FUNCTION_BLOCK FB_MonetTelescopeControl EXTENDS FB_AltAzTelescopeControl IMPLEMENTS I_AltAzTelescope
VAR_INPUT
	fbFocus				: I_Focus;
	fbCovers			: I_MirrorCovers;
	fbBrake				: I_Brake;	
	fbHydraulics   		: I_Hydraulics;
	fbElevation			: REFERENCE TO FB_ElevationControl;
	fbAzimuth			: REFERENCE TO FB_AzimuthControl;
	fbDerotator			: REFERENCE TO FB_DerotatorControl;

	fbPointing			: REFERENCE TO FB_PointingModelForward;
	fbPointingInverse	: REFERENCE TO FB_PointingModelInversion;

	bBrakeClearing		: BOOL	:= TRUE;

	// M6: applied to every commanded elevation move (Goto/Home/Park/PowerOn/Slew, not
	// the computed tracking rate), NOT just _HomeTelescope despite the old name.
	// 5.0 deg/s confirmed correct on-site for MONETS; 10.0 was too fast.
	fElevationMoveVelocity : LREAL := 5.0;
END_VAR
VAR_OUTPUT
	fDerotatorSign		: LREAL := 1.0;	// derotator
	
	fElevationPointingOffset : LREAL;
	fAzimuthPointingOffset : LREAL;
	fElevationPointingOffset2 : LREAL;
	fAzimuthPointingOffset2 : LREAL;
	
	fRightAscensionCurrentSky: LREAL;
	fDeclinationCurrentSky: LREAL;

	fDerotatorVelocity	: LREAL;	// rotational velocity of the derotator
	fElevationVelocity	: LREAL;	// rotational velocity of the elevation
	fAzimuthVelocity	: LREAL;	// rotational velocity of the elevation
END_VAR
VAR
	// M1: internal (non-axis) errors from the Goto/Home/Slew state machines, latched
	// until bReset since bError/nErrorID are otherwise recomputed from the axes every
	// scan and would silently wipe these within the same cycle they're set in.
	bSoftwareError		: BOOL;
	nSoftwareErrorID	: UINT;
	SoftwareErrorEvent	: FB_EventLog;

	// #26 / ADR 0001 option 1: auto-clear a latched bInterrupted if nothing has been
	// requested for a while, since the normal arbitration path can never do it on its
	// own (bReady needs the axes enabled, axis enable needs bInterrupted already clear).
	// Visible, not silent: logged and counted, not just quietly cleared.
	bInterruptedIdle			: BOOL;
	tonInterruptedAutoClear		: TON;
	InterruptedAutoClearEvent	: FB_EventLog;
END_VAR
VAR PERSISTENT
	nInterruptedAutoClearCount	: UDINT;	// how many times auto-clear has fired, ever
END_VAR

// revert fDut1 (set via the Dut1 property, e.g. from an external time bridge over MQTT) to its
// safe 0.0 default if nothing fresh arrives for a while, instead of serving an arbitrarily
// stale UT1-UTC correction forever. FB_AltAzTelescopeControl's own body is never called (this FB
// doesn't call SUPER^() in its main body), so this has to live here rather than up there.
tonDut1Stale(IN := NOT bDut1Received, PT := T#10M);
bDut1Received := FALSE;
IF tonDut1Stale.Q THEN
	fDut1 := 0.0;
END_IF

// get the system time; fJd only follows the clock while the clock is valid (synced, see FB_AstroClock)
fbTime();
IF fbTime.bValid THEN
	fJd := DateTime2JD(fbTime.time_RTCEX2);
END_IF
fLst := CT2LST(telescopeConfig.longitude, fJd);

// without a trustworthy time nothing may be pointed or tracked: refuse through the normal stop path
IF NOT fbTime.bValid AND (bGoto OR bSlew OR bTrack) THEN
	bStop := TRUE;
END_IF

// set reset state either by hardware (key pressed) or by software (set by e.g. tcs)
rtrigReset(CLK := bReset);

IF bReset THEN
	bHorizonError := FALSE; // if reset, the bHorizonError can be switched off
	bSoftwareError := FALSE;
	
	// reset the stages of all statemachine methods
	bInterrupted := TRUE; 
	_HomeTelescope();
	_GotoTelescope();
	_SlewTelescope();
	_ParkTelescope();
	bInterrupted := FALSE;
END_IF

// get error ID, reset if bReset command is set
IF fbAzimuth.Error THEN
	nErrorID := fbAzimuth.nErrorID;
	IF bReset THEN
		fbAzimuth.Reset();
	END_IF
ELSIF fbElevation.bError THEN
	nErrorID := fbElevation.nErrorID;
	IF bReset THEN
		fbElevation.Reset();
	END_IF
ELSIF fbDerotator.bError THEN
	nErrorID := fbDerotator.nErrorID;
	IF bReset THEN
		fbDerotator.Reset();
	END_IF	
ELSIF fbFocus.Error THEN
	nErrorID := fbFocus.ErrorID;
	IF bReset THEN
		fbFocus.Reset();
	END_IF
ELSIF bSoftwareError THEN
	nErrorID := nSoftwareErrorID;
END_IF

// fSlewTime
fSlewTime :=  MAX(MAX(fbElevation.fSlewTime, fbAzimuth.fSlewTime), fbDerotator.fSlewTime);

bError := fbElevation.Error OR
		 fbAzimuth.bError OR
		 fbFocus.Error OR
		 fbDerotator.bError OR
		 bSoftwareError;
			
IF bError THEN
	bTrack := 	FALSE;
	bGoto := 	FALSE;
	bSlew := 	FALSE;
	fbElevation.Enable := FALSE;
	fbAzimuth.Enable := FALSE;
	fbDerotator.Enable := FALSE;
ELSE
	nErrorID := 0;
END_IF

IF fbElevation.bError THEN
	fbElevation.Enable := FALSE;
	fbAzimuth.Enable := FALSE;
	fbDerotator.Enable := FALSE;
	fbBrake.CloseBrake();
END_IF

eq2hor(
	ra := fRightAscension,
	dec := fDeclination,
	lon := telescopeConfig.longitude,
	lat := telescopeConfig.latitude,
	altitude := telescopeConfig.altitude,
	JD := fJd + fTimeOffset,
	dut1 := fDut1,
	refract_to_observed := TRUE,
	// refract := FALSE,
	alt => fElevationCalc,
	az => fAzimuthCalc,
	ha => fHourAngleCalc);

// apply pointing model
fbPointing(
	fAzimuth			:= fAzimuthCalc,
	fElevation			:= fElevationCalc,
	fAzimuthOffset		=> fAzimuthPointingOffset,
	fElevationOffset	=> fElevationPointingOffset
);
fElevationCalc := fElevationCalc + fElevationPointingOffset + fElevationOffset;
// F_AzimuthOffsetOnAxis: fAzimuthOffset / COS(elevation), bounded near the zenith (BROTLib#27)
fAzimuthCalc := fAzimuthCalc + fAzimuthPointingOffset + F_AzimuthOffsetOnAxis(fAzimuthOffset, fElevationCalc);

// calculate derotator position 
fDerotatorCalc := F_DerotatorPosition2(fAzimuthCalc, fElevationCalc, telescopeConfig.latitude, fDerotatorSign)  + fDerotatorOffset;

// calculate velocities
fDerotatorVelocity := F_Derotatorvelocity(fAzimuthCalc, fElevationCalc, telescopeConfig.latitude, fDerotatorSign);
fElevationVelocity := F_Elevationvelocity(fAzimuthCalc, telescopeConfig.latitude);
fAzimuthVelocity := F_Azimuthvelocity(fElevationCalc, fAzimuthCalc, telescopeConfig.latitude);

IF (fAzimuthCalc > 310.0 AND fAzimuthVelocity > 0.0) OR (fAzimuthCalc > 440.0) THEN
	fAzimuthCalc := fAzimuthCalc - 360.0;
ELSIF (fAzimuthCalc < 80.0 AND fAzimuthVelocity < 0.0) OR (fAzimuthCalc < -50.0) THEN
	fAzimuthCalc := fAzimuthCalc + 360.0;
END_IF

IF (fDerotatorCalc > 290.0 AND fDerotatorVelocity > 0.0) OR (fDerotatorCalc > 380.0) THEN
	fDerotatorCalc := fDerotatorCalc - 360.0;
ELSIF (fDerotatorCalc < 20.0 AND fDerotatorVelocity < 0.0) OR (fDerotatorCalc < -70.0) THEN
	fDerotatorCalc := fDerotatorCalc + 360.0;
END_IF

// get current coordinates	
fAzimuthCurrent := fbAzimuth.fActualPosition;
fElevationCurrent := fbElevation.fActualPosition;
fDerotatorCurrent := fbDerotator.fActualPosition;

// apply inverse pointing model
fbPointingInverse(
	fAzimuth			:= fAzimuthCurrent,
	fElevation			:= fElevationCurrent,
	fAzimuthOffset  	=> fAzimuthPointingOffset2,
	fElevationOffset	=> fElevationPointingOffset2
);
fAzimuthCurrentSky := fAzimuthCurrent - fAzimuthPointingOffset2;
fElevationCurrentSky := fElevationCurrent - fElevationPointingOffset2;

// add offsets
//fElevationCurrent := fElevationCurrentSky - fElevationOffset;
//fAzimuthCurrent := fAzimuthCurrentSky - fAzimuthOffset / COS(fElevationCalc * d2r);

// calculate equatorial coordinates
hor2eq(alt := fElevationCurrentSky - fElevationOffset,
		az := fAzimuthCurrentSky - F_AzimuthOffsetOnAxis(fAzimuthOffset, fElevationCurrent),	// M7: was fElevationCalc
		jd := fJd,
		dut1 := fDut1,
		lat := telescopeConfig.latitude,
		lon := telescopeConfig.longitude,
		altitude := telescopeConfig.altitude,
		alt_is_observed := TRUE,
		// refract := FALSE,
		ra => fRightAscensionCurrent,
		dec => fDeclinationCurrent,
		ha => fHourAngleCurrent);	// M13: was never assigned, HA_ICRS telemetry was stuck at 0.0
hor2eq(alt := fElevationCurrentSky,
		az := fAzimuthCurrentSky,
		jd := fJd,
		dut1 := fDut1,
		lat := telescopeConfig.latitude,
		lon := telescopeConfig.longitude,
		altitude := telescopeConfig.altitude,
		alt_is_observed := TRUE,
		ra => fRightAscensionCurrentSky,
		dec => fDeclinationCurrentSky);
	
// If the Telescope dips under the fHorizon (e.g. while tracking, stop and gohome)
IF fbElevation.Calibrated AND fElevationCurrent < (fHorizon+0.2) THEN
	IF NOT bStopped AND NOT bGoHome THEN
		bStop := TRUE;
	ELSE
		bGoHome := TRUE;
	END_IF
END_IF
		
tpPowerOnWarning(IN := bPower OR (NOT fbElevation.bEnable AND fbBrake.BrakeOpen), PT := T#250MS);

tonPowerTimeout(IN := TCS_command = E_TCSCommand.no_command AND NOT bIsParked, PT := T#12H);
tonCommandTimeout();
IF tonPowerTimeout.Q AND NOT bIsParked THEN
	bPark := TRUE;
END_IF
		
// #26 / ADR 0001 option 1: bInterrupted otherwise cannot clear itself once latched with
// nothing pending (see specs/design/telescopecontrol-command-arbitration.md); auto-clear
// after a few seconds of true idle (no error, nothing requested), logged and counted so
// it's visible rather than a silent recovery. TUNE PT if this fires too eagerly/late on
// site.
bInterruptedIdle := bInterrupted AND NOT bError AND
	NOT (bPower OR bPark OR bGoHome OR bGoto OR bSlew OR bTrack);
tonInterruptedAutoClear(IN := bInterruptedIdle, PT := T#5S);
IF tonInterruptedAutoClear.Q THEN
	bInterrupted := FALSE;
	nInterruptedAutoClearCount := nInterruptedAutoClearCount + 1;
END_IF
InterruptedAutoClearEvent(
	Trigger 		:= tonInterruptedAutoClear.Q,
	Level 			:= ADSLOG_MSGTYPE_WARN,
	FormatString 	:= 'bInterrupted auto-cleared after idle timeout (count: %s)',
	OnMessage 		:= UDINT_TO_STRING(nInterruptedAutoClearCount),
	Comm 			:= fbComm);

// set TCS_command according to state variables ordered by precedence
// Stop outranks everything, including a running power-on
IF bStop THEN
	bTrack := FALSE;
	
	// If the stop is during a power-on or a movement, reset the stage of the movement first
	IF bPower THEN
		bPower := FALSE;
		_PowerOn();
	END_IF
	IF bPark THEN
		bPark := FALSE;
		_ParkTelescope();
	ELSIF bGoto THEN
		bGoto := FALSE;
		_GotoTelescope();
	ELSIF bSlew THEN
		bSlew := FALSE;
		_SlewTelescope();
	ELSIF bGoHome THEN
		bGoHome := FALSE;
		_HomeTelescope();
	END_IF
	TCS_command := E_TCSCommand.stop;
	
ELSIF bPower THEN
	TCS_command := E_TCSCommand.poweron;
	
ELSIF bPark THEN
	bTrack := FALSE;
	// M2: emergency park bypasses the bReady/bBusy gating below entirely, since bReady
	// requires NOT bError and would otherwise make park unreachable during an error.
	IF bError THEN
		bInterrupted := FALSE;
		TCS_command := E_TCSCommand.park;
	// If lower presedence commands are ongoing, let them know they are interupted
	ELSIF bGoto OR bSlew OR bGoHome THEN
		bGoHome := FALSE;
		bGoto := FALSE;
		bSlew := FALSE;
		bInterrupted := TRUE;
		_HomeTelescope();
		_GotoTelescope();
		_SlewTelescope();

	ELSE
		IF bReady AND NOT bBusy THEN
			bInterrupted := FALSE;
			TCS_command := E_TCSCommand.park;
		END_IF
	END_IF
	
ELSIF bGoHome THEN
	bTrack := FALSE;
	// If lower presedence commands are ongoing, let them know they are interupted
	IF bGoto OR bSlew THEN
		bGoto := FALSE;
		bSlew := FALSE;
		bInterrupted := TRUE;
		_GotoTelescope();
		_SlewTelescope();
		
	ELSE
		IF bReady AND NOT bBusy AND bStopped THEN
			bInterrupted := FALSE;
			TCS_command := E_TCSCommand.gohome;
		END_IF
	END_IF
	
	
ELSIF bGoto THEN
	bTrack := FALSE;
	// If lower presedence commands are ongoing, let them know they are interupted
	IF bSlew THEN
		bSlew := FALSE;
		bInterrupted := TRUE;
		_SlewTelescope();
	ELSE
		IF bReady AND NOT bBusy THEN
			bInterrupted := FALSE;
			TCS_command := E_TCSCommand.goto;
		END_IF
	END_IF
		
ELSIF bSlew THEN
	bTrack := FALSE;
	IF bReady AND NOT bBusy THEN
		TCS_command := E_TCSCommand.slew;
	END_IF
	
ELSIF bTrack THEN
	IF bReady AND NOT bBusy THEN
		TCS_command := E_TCSCommand.track;
	END_IF
	
ELSE
	TCS_command := E_TCSCommand.no_command;
	fbElevation.bMoveAxis := FALSE;
	fbAzimuth.bMoveAxis := FALSE;
	fbDerotator.bMoveAxis := FALSE;
	fbElevation.bTracking := FALSE;
	fbAzimuth.bTracking := FALSE;
	fbDerotator.bTracking := FALSE;
END_IF

IF TCS_command = E_TCSCommand.poweron THEN
	_PowerOn();
	tonCommandTimeout(IN := TCS_command = E_TCSCommand.poweron, PT := T#12H);
	TCSCTOEvent.OnMessage := 'POWER';
ELSIF TCS_command = E_TCSCommand.stop THEN
	_StopTelescope();
	tonCommandTimeout(IN := TCS_command = E_TCSCommand.stop, PT := T#2S);
	TCSCTOEvent.OnMessage := 'STOP';
ELSIF TCS_command = E_TCSCommand.park THEN
	_ParkTelescope();
	tonCommandTimeout(IN := TCS_command = E_TCSCommand.park, PT := T#2M);
	TCSCTOEvent.OnMessage := 'PARK';
ELSIF TCS_command = E_TCSCommand.gohome THEN
	_HomeTelescope();
	tonCommandTimeout(IN := TCS_command = E_TCSCommand.gohome, PT := T#2M);
	TCSCTOEvent.OnMessage := 'GOHOME';
ELSIF TCS_command = E_TCSCommand.goto THEN
	_GotoTelescope();
	tonCommandTimeout(IN := TCS_command = E_TCSCommand.goto, PT := T#2M);
	TCSCTOEvent.OnMessage := 'GOTO';
ELSIF TCS_command = E_TCSCommand.slew THEN
	_SlewTelescope();
	tonCommandTimeout(IN := TCS_command = E_TCSCommand.slew, PT := T#2M);
	TCSCTOEvent.OnMessage := 'SLEW';
ELSIF TCS_command = E_TCSCommand.track THEN
	_TrackTelescope();
	tonCommandTimeout(IN := TCS_command = E_TCSCommand.track, PT := T#12H);
	TCSCTOEvent.OnMessage := 'TRACK';
ELSE
	// disable command timeout
	tonCommandTimeout(IN := FALSE);
	TCSCTOEvent.OnMessage := 'NOCOMMAND';
END_IF
 
bSlewing := NOT bTracking AND (fbElevation.fbAxis.InMotion OR fbElevation.fbAxis.InRamp OR
			fbAzimuth.fbAxis.InMotion OR fbAzimuth.fbAxis.InRamp OR
			fbDerotator.fbAxis.InMotion OR fbDerotator.fbAxis.InRamp);

// signal must be stable for 5500MS
tonTrackingDelay(in := fbElevation.fbAxis.isTracking AND 
			fbAzimuth.fbAxis.isTracking AND
			fbDerotator.fbAxis.isTracking,PT :=T#5500MS, Q => bTracking);
			
bStopped :=  (NOT fbElevation.bEnable OR fbElevation.fbAxis.StandStill) AND 
			(NOT fbAzimuth.bEnable OR fbAzimuth.fbAxis.StandStill) AND
			(NOT fbDerotator.bEnable OR fbDerotator.fbAxis.StandStill);
			
bHomed := fbElevation.Calibrated AND
			fbAzimuth.Calibrated AND
			fbFocus.Calibrated AND
			fbDerotator.Calibrated;
			
bReady := bHomed AND 
	fbCovers.Opened AND 
	fbElevation.bEnable AND
	fbAzimuth.bEnable AND
	fbDerotator.bEnable AND fbBrake.BrakeOpen AND 
    NOT bError;

bBusy := fbElevation.fbAxis.Busy OR
		fbAzimuth.fbAxis.Busy OR
		fbDerotator.fbAxis.Busy OR
		fbFocus.Busy;

(* STATUS STATES*)
//fReadyState (see also _PowerOn and _ParkTelescope calls above)
IF bError THEN
	fReadyState := -1.0;
ELSIF bPower THEN
	fReadyState := 0.7;
ELSIF bIsParked THEN
	fReadyState := 0.0;
ELSIF bPark THEN
	fReadyState := 0.3;
ELSIF bReady THEN
	fReadyState := 1.0;	
ELSE
	fReadyState := -2.0;	
END_IF

//MotionState
IF bStopped THEN
	nMotionState := 0;
ELSIF bSlewing OR bBusy THEN
	nMotionState := 1;
ELSIF bTracking THEN
	nMotionState := 8;
END_IF

// unset the STOP command if telescope is already stopped
IF bStopped THEN
	bStop := FALSE;
END_IF
	
IF NOT bError THEN
	bReset := FALSE;
END_IF

IF bEstopTriggered THEN
	fbElevation.Enable := FALSE;
	fbAzimuth.Enable := FALSE;
	fbDerotator.Enable := FALSE;
END_IF

// send telemetry
IF bSlewing OR bTrack OR bTracking THEN
	tonMQTTTimer.PT := T#500MS; // M13: was "every second", actually twice a second while moving
ELSE
	tonMQTTTimer.PT := T#1000MS; // M13: was "every five seconds", actually every second otherwise
END_IF
tonMQTTTimer(IN:=TRUE);
IF tonMQTTTimer.Q THEN
	tonMQTTTimer(IN:=FALSE);
	_SendTelemetry();
END_IF


(* Event function blocks start here. *)
TCSpowerEvent(	Trigger := bPowerFailure, 
				Level := ADSLOG_MSGTYPE_ERROR,
				FormatString := 'power %s',
				//OnMessage := 'Failure',
				OffMessage := 'OK', 
				Comm := fbComm);

TCSgohomeEvent(	Trigger := bGoHome, 
				Level := ADSLOG_MSGTYPE_HINT,
				FormatString := 'GOHOME %s',
				OnMessage := 'commencing',
				OffMEssage := 'completed', 
				Comm := fbComm);
TCSparkEvent(	Trigger := bPark, 
				Level := ADSLOG_MSGTYPE_HINT,
				FormatString := 'PARK %s',
				OnMessage := 'commencing',
				OffMEssage := 'completed', 
				Comm := fbComm);
TCSgotoEvent(	Trigger := bGoto, 
				Level := ADSLOG_MSGTYPE_HINT,
				FormatString := 'GOTO %s',
				OnMessage := 'commencing',
				OffMEssage := 'completed', 
				Comm := fbComm);
TCStrackEvent(	Trigger := bTrack, 
				Level := ADSLOG_MSGTYPE_HINT,
				FormatString := 'TRACK %s',
				OnMessage := 'commencing',
				OffMEssage := 'completed', 
				Comm := fbComm);
TCSstopEvent(	Trigger := bStop, 
				Level := ADSLOG_MSGTYPE_WARN,
				FormatString := 'STOP %s',
				OnMessage := 'commencing',
				OffMEssage := 'completed',
				OffLevel := ADSLOG_MSGTYPE_HINT, 
				Comm := fbComm);
TCStargetHorizonEvent(	Trigger := fElevationCalc<fHorizon,
				Level := ADSLOG_MSGTYPE_WARN,
				FormatString := '%s',
				OnMessage := 'Target below safe horizon',
				OffMEssage := '', 
				Comm := fbComm);
TCSreadyEvent(	Trigger := bPower AND bReady, 
				Level := ADSLOG_MSGTYPE_HINT,
				FormatString := '%s',
				OnMessage := 'STELLA1 startup finished', 
				Comm := fbComm);
TCSCTOEvent(	Trigger := tonCommandTimeout.Q,
				Level := ADSLOG_MSGTYPE_WARN,
				FormatString := 'A timeout occurred during %s command!',
				OnMessage := 'NOCOMMAND',
				Comm := fbComm);
SoftwareErrorEvent(	Trigger := bSoftwareError,
				Level := ADSLOG_MSGTYPE_ERROR,
				FormatString := 'Internal command error, ID: %s',
				OnMessage := UINT_TO_STRING(nSoftwareErrorID),
				OffMessage := 'cleared',
				OffLevel := ADSLOG_MSGTYPE_HINT,
				Comm := fbComm);

METHOD PRIVATE _GotoTelescope : USINT
VAR_INPUT
END_VAR
VAR
	GoToEvent		: FB_Eventlog;
	commandTimeout	: TON;
END_VAR
VAR_STAT
	nStage			: USINT := 0;
	nLastStage		: USINT := 101;
END_VAR
_GotoTelescope := nStage;
commandTimeout(IN := nStage < 100, PT := T#600S);
IF commandTimeout.Q THEN
	bError := TRUE;
	nErrorID := 16#10;
	bSoftwareError := TRUE;
	nSoftwareErrorID := 16#10;
	bGoto := FALSE;
	nStage := 0;
	RETURN;
END_IF

IF fElevationCalc<2.0 THEN
	bError := TRUE;
	nErrorID := 16#15;
	bSoftwareError := TRUE;
	nSoftwareErrorID := 16#15;
	bGoto := FALSE;
	nStage := 0;
	RETURN;
END_IF

// M7: near zenith COS(elevation) -> 0, so any nonzero fAzimuthOffset blows up into a
// huge azimuth (see the offset divisions elsewhere in this FB). 89.5 matches the
// existing tracking cutoff (_TrackTelescope: fElevationCurrent > 89.5).
IF fElevationCalc>89.5 THEN
	bError := TRUE;
	nErrorID := 16#16;
	bSoftwareError := TRUE;
	nSoftwareErrorID := 16#16;
	bGoto := FALSE;
	nStage := 0;
	RETURN;
END_IF

IF bReset OR bError OR bInterrupted THEN
	nStage := 0;
	RETURN;
END_IF

CASE nStage OF
	0:	
		IF bReady AND NOT bBusy THEN
			nStage := 10;
		END_IF
	10:
		IF fbElevation.Tracking = TRUE OR fbAzimuth.Tracking = TRUE OR fbDerotator.Tracking = TRUE THEN
			fbElevation.Tracking := FALSE;
			fbAzimuth.Tracking := FALSE;
			fbDerotator.Tracking := FALSE;
		ELSE
			nStage := 25;
		END_IF				
	25:	
		fbElevation.Position := fElevationCalc;
		fbAzimuth.Position := fAzimuthCalc;
		fbDerotator.Position := fDerotatorCalc;
		fbDerotator.Velocity := 10.0;
		fbElevation.Velocity := fElevationMoveVelocity;
		fbAzimuth.Velocity := 10.0;
		
		fbElevation.MoveAxis := TRUE;
		fbAzimuth.MoveAxis := TRUE;
		fbDerotator.MoveAxis := TRUE;
		IF fbElevation.Busy AND
			fbAzimuth.Busy AND
			fbDerotator.Busy THEN
				nStage := 50;
		END_IF
	50:
		IF NOT fbElevation.Busy AND fbElevation.MoveDone THEN
			fbElevation.MoveAxis := FALSE;
		END_IF
		IF NOT fbAzimuth.Busy AND fbAzimuth.MoveDone THEN
			fbAzimuth.MoveAxis := FALSE;
		END_IF
		IF NOT fbDerotator.Busy AND fbDerotator.MoveDone THEN
			fbDerotator.MoveAxis := FALSE;
		END_IF
		IF NOT fbElevation.MoveAxis AND 
           NOT fbAzimuth.MoveAxis AND 
		   NOT fbDerotator.MoveAxis THEN
		   nStage := 75;
		END_IF
	75:
		IF NOT bSlewing AND bStopped THEN // all axis standstill
			nStage := 100;
		END_IF
	100:
		fbElevation.MoveAxis := FALSE;
		fbAzimuth.MoveAxis := FALSE;
		fbDerotator.MoveAxis := FALSE;
		fAzimuth := fAzimuthCalc;
		fElevation := fElevationCalc;
		bGoto := FALSE;
		// enable automatic tracking
		bTrack := bAutoTrack;
		nStage := 0;
END_CASE
GoToEvent(Trigger := nStage > nLastStage, FormatString := 'GoTo progress: %s', OnMessage := USINT_TO_STRING(nStage), comm := fbComm);
nLastStage := nStage;
END_METHOD

METHOD PRIVATE _HomeTelescope : BOOL
VAR_INPUT
END_VAR
VAR
    HomeEvent        : FB_Eventlog;
    commandTimeout    : TON;
END_VAR
// reset/interrupt aborts the homing without moving anything, like the other stage methods
IF bReset OR bError OR bInterrupted THEN
    commandTimeout(IN := FALSE);
    RETURN;
END_IF

commandTimeout(IN := NOT _HomeTelescope, PT := T#600S);
IF commandTimeout.Q THEN
    bError := TRUE;
    nErrorID := 16#30;
    bSoftwareError := TRUE;
    nSoftwareErrorID := 16#30;
    _HomeTelescope :=TRUE;
END_IF

// only move while a home command is active (Stop/Park/Reset call this with bGoHome cleared to abort it)
IF bGoHome AND bReady AND bStopped AND NOT bBusy AND NOT bTracking THEN
    fbElevation.Velocity := fElevationMoveVelocity;
    fbElevation.Position := telescopeConfig.elevationHome;
    fbElevation.MoveAxis := TRUE;
    fbAzimuth.Velocity := 10.0;
    fbAzimuth.Position := telescopeConfig.azimuthHome;
    fbAzimuth.MoveAxis := TRUE;
    fbDerotator.Velocity := 10.0;
    fbDerotator.Position := telescopeConfig.derotatorHome;
    fbDerotator.MoveAxis := TRUE;    
END_IF

IF fbElevation.MoveDone AND 
    fbAzimuth.MoveDone AND 
    fbDerotator.MoveDone THEN
    bGoHome := FALSE;
    fElevation := fElevationCurrent;
    fAzimuth := fAzimuthCurrent;
    _HomeTelescope := TRUE;
ELSE
    _HomeTelescope := FALSE;
END_IF

HomeEvent(Trigger := _HomeTelescope, 
            Level := ADSLOG_MSGTYPE_HINT,
            FormatString := '%s',
            OnMessage := 'Telescope is homed.', comm := fbComm);
END_METHOD

METHOD PRIVATE _ParkTelescope : USINT
VAR_INPUT
END_VAR
VAR
	ParkEvent	: FB_Eventlog;
	rtrigError	: R_TRIG;	// M2: reset the stage only on the rising edge of bError, not every scan
END_VAR
VAR_STAT
	nStage		: USINT := 0;
	nLastStage	: USINT := 101;
END_VAR
_ParkTelescope := nStage;
IF bReset OR bStop OR bInterrupted THEN
	nStage := 0;
	RETURN;
END_IF
// M2: bError does NOT return early here, unlike the other state machines: stage 0's
// "emergency park" branch below is the safe-state response to bError and must run.
// Only force the stage back to 0 on the rising edge, so the emergency branch can still
// progress through its own stages (80 -> 100) on later scans while bError stays TRUE.
rtrigError(CLK := bError);
IF rtrigError.Q THEN
	nStage := 0;
END_IF
IF bIsParked THEN
	nStage := 100;
END_IF
CASE nStage OF
	0: 
		bGoHome := 	FALSE;
		bTrack := 	FALSE;
		bGoto := 	FALSE;
		bSlew := 	FALSE;
		fbFocus.Position := telescopeConfig.focusPark;
		IF bError THEN // emergency park
			fbBrake.CloseBrake();
			fbElevation.Enable := FALSE;
			fbAzimuth.Enable := FALSE;
			fbDerotator.Enable := FALSE;	
			fbCovers.Close();	
			nStage := 80;
		ELSE
			nStage := 10;
		END_IF
	10:
		IF fbElevation.Tracking = TRUE OR fbAzimuth.Tracking = TRUE OR fbDerotator.Tracking = TRUE THEN
			fbElevation.Tracking := FALSE;
			fbAzimuth.Tracking := FALSE;
			fbDerotator.Tracking := FALSE;
		ELSE
			nStage := 20;
		END_IF		
	20:
		fbElevation.Position := telescopeConfig.elevationPark;
		fbElevation.Velocity := fElevationMoveVelocity;
		fbElevation.MoveAxis := TRUE;
		fbAzimuth.Position := telescopeConfig.azimuthPark;
		fbAzimuth.Velocity := 10;
		fbAzimuth.MoveAxis := TRUE;
		fbDerotator.Position := telescopeConfig.derotatorPark;
		fbDerotator.Velocity := 10.0;
		fbDerotator.MoveAxis := TRUE;
		IF fbElevation.Busy AND
			fbAzimuth.Busy AND
			fbDerotator.Busy THEN
				nStage := 40;
		END_IF
	40:
		IF fbElevation.MoveDone THEN
			fbElevation.MoveAxis := FALSE;
		END_IF
		IF fbAzimuth.MoveDone THEN
			fbAzimuth.MoveAxis := FALSE;
		END_IF
		IF fbDerotator.MoveDone THEN
			fbDerotator.MoveAxis := FALSE;
		END_IF
		IF NOT bSlewing THEN // all axis standstill
			nStage := 60;
		END_IF
	60:
		IF NOT fbElevation.Enable AND NOT fbAzimuth.Enable AND NOT fbDerotator.Enable THEN
			nStage := 80;
		END_IF

		IF bStopped THEN
			fbElevation.Enable := FALSE;
			fbAzimuth.Enable := FALSE;
			fbDerotator.Enable := FALSE;
		END_IF
		
		fbElevation.bMoveAxis := FALSE;
		fbAzimuth.bMoveAxis := FALSE;
		fbDerotator.bMoveAxis := FALSE;
	80:
		IF fbElevation.Enable OR fbAzimuth.Enable OR fbDerotator.Enable THEN
			nStage := 60;
		END_IF
		IF NOT fbBrake.BrakeOpen THEN
			fbCovers.Close();
			fbHydraulics.Enable := FALSE;
		END_IF
		IF fbCovers.Closed THEN
			nStage := 100;
		END_IF
	100:
			bIsParked := TRUE;
			bPark := FALSE;
			_ParkTelescope := 100;
			nStage := 0;	
END_CASE
ParkEvent(Trigger := nStage > nLastStage, FormatString := 'Parking progress: %s', OnMessage := USINT_TO_STRING(nStage), comm := fbComm);
nLastStage := nStage;
END_METHOD

METHOD PRIVATE _PowerOn : BOOL
VAR_INPUT
END_VAR
VAR_STAT
	nStage		: USINT := 0;
	nLastStage	: USINT := 101;
END_VAR
IF NOT bBrakeClearing THEN
	bPowerFailure := TRUE;
	TCSpowerEvent.OnMessage := 'failure: brake clearing not set';
	bPower := FALSE;
ELSIF bError THEN
	bPowerFailure := TRUE;
	TCSpowerEvent.OnMessage := 'Generic error during power on occurred.';
	bPower := FALSE;
ELSE
	bPowerFailure := FALSE;		
END_IF

IF bReset OR bError OR bStop OR bInterrupted THEN
	nStage := 0;
	// abort without leaving the last written axis commands set
	fbElevation.MoveAxis := FALSE;
	fbElevation.HomeAxis := FALSE;
	fbAzimuth.MoveAxis := FALSE;
	fbAzimuth.HomeAxis := FALSE;
	fbDerotator.MoveAxis := FALSE;
	fbDerotator.HomeAxis := FALSE;
	fbFocus.HomeAxis := FALSE;
	RETURN;
END_IF

CASE nStage OF
	0:
		_PowerOn := FALSE;
		// COVER MUST BE OPENED FOR A SUCCESSFUL WAKE & SHAKE COMMAND!
		// unconditional by design: does not consult bCoverAutoOpen (see CoverAutoOpen.Set)
		fbCovers.Open();
		IF bMainReady AND fbCovers.Opened THEN
			nStage := 10;
		END_IF
		
	10:
		fbElevation.Enable := TRUE;
		fbAzimuth.Enable := TRUE;
		fbDerotator.Enable := TRUE;
		
		IF fbElevation.Ready AND NOT fbElevation.Calibrated THEN
			fbElevation.HomeAxis := TRUE;
		END_IF
		
		IF fbAzimuth.Ready AND NOT fbAzimuth.Calibrated THEN
			fbAzimuth.HomeAxis := TRUE;
		END_IF
		
		// enable derotator
		IF fbElevation.Ready THEN
			fbDerotator.HomeAxis := fbDerotator.Ready AND NOT fbDerotator.Calibrated;
		END_IF
		
		// start calibration of focus after elevation has been calibrated
		// this avoids imbalance by the M2 mirror on the elvation during its calibration
		IF fbElevation.Calibrated AND NOT fbFocus.Calibrated THEN
			fbFocus.Enable := TRUE;
			fbFocus.HomeAxis := TRUE;
		END_IF
	
		IF fbCovers.Opened AND fbElevation.Calibrated AND fbAzimuth.Calibrated AND fbDerotator.Calibrated AND fbFocus.Calibrated AND
			bReady AND bStopped AND NOT bBusy AND NOT bTracking THEN
			nStage := 30;
		END_IF
		
	30:
		fbElevation.Velocity := fElevationMoveVelocity;
		fbElevation.Position := telescopeConfig.elevationHome;
		fbElevation.MoveAxis := TRUE;
		fbAzimuth.Velocity := 10.0;
		fbAzimuth.Position := telescopeConfig.azimuthHome;
		fbAzimuth.MoveAxis := TRUE;
		fbDerotator.Velocity := 10.0;
		fbDerotator.Position := telescopeConfig.derotatorHome;
		fbDerotator.MoveAxis := TRUE;	
		
		IF fbElevation.MoveDone AND 
			fbAzimuth.MoveDone AND 
			fbDerotator.MoveDone THEN
			nStage := 100;
		END_IF
			
	100:
		bPower := FALSE;
		fElevation := fElevationCurrent;
		fAzimuth := fAzimuthCurrent;
		_PowerOn := TRUE;
		bIsParked := FALSE;
		nStage := 0;
	
END_CASE
END_METHOD

METHOD _SendTelemetry : BOOL
VAR_INPUT
END_VAR
SUPER^._PublishTelemetry();

fbComm.Publish('telescope', 'dome', 'TELESCOPE.READY_STATE',	LREAL_TO_STRING(fReadyState));
fbComm.Publish('telescope', 'dome', 'TELESCOPE.MOTION_STATE',	LREAL_TO_STRING(nMotionState));
fbComm.Publish('telescope', 'dome', 'TELESCOPE.INTERRUPTED_AUTO_CLEAR_COUNT', UDINT_TO_STRING(nInterruptedAutoClearCount));

// INFO, CONFIG.MOUNTOPTIONS/MOUNT, STATUS.GLOBAL, OBJECT.INSTRUMENTAL.ALT/AZ and the static
// OBJECT.EQUATORIAL.EPOCH/EQUINOX/RA_PM/DEC_PM/RA_RATE/DEC_RATE fields used to be republished
// here too, byte-identical to what SUPER^._PublishTelemetry() above already sends under the same
// field names from the same source variables -- removed as pure duplication (#22).
//
// OBJECT.EQUATORIAL.RA_ICRS/DEC_ICRS kept even though pybrotlib's schema (the Python MQTT
// consumer, BROTLib/pyBROT src/pybrotlib/telemetry.py) has no such field under
// object.equatorial -- only object.equatorial.ra/dec, which SUPER already publishes with the
// same value -- so this specific publish looks like dead weight for that consumer. Not removing
// it here anyway: Telegraf/InfluxDB ingests the raw MQTT line independent of pybrotlib's schema,
// so something else could still depend on this exact field name landing in Influx. (For contrast,
// POSITION.EQUATORIAL.RA_ICRS/DEC_ICRS -- a different field, published further down -- *is* in
// pybrotlib's schema and is a real, actively consumed field.)
//
// OBJECT.HORIZONTAL.ALT/AZ below is also kept even though SUPER publishes those same field names:
// SUPER's version is conditional on bSlew (fElevation/fAzimuth vs fElevationCalc/fAzimuthCalc);
// this unconditional republish runs after it and is what has actually been on the wire -- changing
// that is a behavior change, not a dedup.

// EQUATORIAL
// all angles in the telemetry are degrees, RA included, like the rightascension command (BROTLib#37)
fbComm.Publish('telescope', 'dome', 'OBJECT.EQUATORIAL.RA_ICRS', LREAL_TO_STRING(fRightAscension));
fbComm.Publish('telescope', 'dome', 'OBJECT.EQUATORIAL.DEC_ICRS', LREAL_TO_STRING(fDeclination));

// HORIZONTAL
fbComm.Publish('telescope', 'dome', 'OBJECT.HORIZONTAL.ALT', LREAL_TO_STRING(fElevationCalc));
fbComm.Publish('telescope', 'dome', 'OBJECT.HORIZONTAL.AZ', LREAL_TO_STRING(fAzimuthCalc));

(* POINTING *)
fbComm.Publish('telescope', 'dome', 'POINTING.SLEWTIME', LREAL_TO_STRING(fSlewtime));
fbComm.Publish('telescope', 'dome', 'POINTING.OFFSETS.ALT', LREAL_TO_STRING(fElevationPointingOffset));
fbComm.Publish('telescope', 'dome', 'POINTING.OFFSETS.AZ', LREAL_TO_STRING(fAzimuthPointingOffset));

(*POSITION*)
//LOCAL
fbComm.Publish('telescope', 'dome', 'POSITION.LOCAL.SIDEREAL_TIME', LREAL_TO_STRING(fLst));
fbComm.Publish('telescope', 'dome', 'POSITION.LOCAL.JD', LREAL_TO_STRING(fJd));
fbComm.Publish('telescope', 'dome', 'POSITION.LOCAL.LATITUDE', LREAL_TO_STRING(telescopeConfig.latitude));
fbComm.Publish('telescope', 'dome', 'POSITION.LOCAL.LONGITUDE', LREAL_TO_STRING(telescopeConfig.longitude));
fbComm.Publish('telescope', 'dome', 'POSITION.LOCAL.HEIGHT', LREAL_TO_STRING(telescopeConfig.altitude));

// INSTRUMENTAL
// > ALT
// POWER_STATE
IF fbElevation.Enable THEN
	fbComm.Publish('telescope', 'dome', 'POSITION.INSTRUMENTAL.ALT.POWER_STATE', '1.0');
ELSE
	fbComm.Publish('telescope', 'dome', 'POSITION.INSTRUMENTAL.ALT.POWER_STATE', '0.0');
END_IF
//REFERENCED
IF fbElevation.Calibrated THEN
	fbComm.Publish('telescope', 'dome', 'POSITION.INSTRUMENTAL.ALT.REFERENCED', '1.0');
ELSE
	fbComm.Publish('telescope', 'dome', 'POSITION.INSTRUMENTAL.ALT.REFERENCED', '0.0');
END_IF
//ERROR_STATE
IF fbElevation.Error THEN
	fbComm.Publish('telescope', 'dome', 'POSITION.INSTRUMENTAL.ALT.ERROR_STATE', UDINT_TO_STRING(fbElevation.ErrorID));
ELSE
	fbComm.Publish('telescope', 'dome', 'POSITION.INSTRUMENTAL.ALT.ERROR_STATE', '0');
END_IF
//MOTION_STATE
IF fbElevation.Busy THEN
	IF fbElevation.isTracking THEN
		fbComm.Publish('telescope', 'dome', 'POSITION.INSTRUMENTAL.ALT.MOTION_STATE', '8');
	ELSE
		fbComm.Publish('telescope', 'dome', 'POSITION.INSTRUMENTAL.ALT.MOTION_STATE', '1');
	END_IF
ELSE
	fbComm.Publish('telescope', 'dome', 'POSITION.INSTRUMENTAL.ALT.MOTION_STATE', '0');
END_IF
fbComm.Publish('telescope', 'dome', 'POSITION.INSTRUMENTAL.ALT.REALPOS', LREAL_TO_STRING(fElevationCurrent-fElevationOffset));
fbComm.Publish('telescope', 'dome', 'POSITION.INSTRUMENTAL.ALT.CURRPOS', LREAL_TO_STRING(fElevationCurrent));
fbComm.Publish('telescope', 'dome', 'POSITION.INSTRUMENTAL.ALT.TARGETPOS', LREAL_TO_STRING(fbElevation.Position));
fbComm.Publish('telescope', 'dome', 'POSITION.INSTRUMENTAL.ALT.CURRSPEED', LREAL_TO_STRING(fbElevation.Velocity));
fbComm.Publish('telescope', 'dome', 'POSITION.INSTRUMENTAL.ALT.TARGETDISTANCE', LREAL_TO_STRING(ABS(fElevationCurrent-fbElevation.Position)));
fbComm.Publish('telescope', 'dome', 'POSITION.INSTRUMENTAL.ALT.OFFSET', LREAL_TO_STRING(fElevationOffset));

// > AZ
// POWER_STATE
IF fbAzimuth.Enable THEN
	fbComm.Publish('telescope', 'dome', 'POSITION.INSTRUMENTAL.AZ.POWER_STATE', '1.0');
ELSE
	fbComm.Publish('telescope', 'dome', 'POSITION.INSTRUMENTAL.AZ.POWER_STATE', '0.0');
END_IF
//REFERENCED
IF fbAzimuth.Calibrated THEN
	fbComm.Publish('telescope', 'dome', 'POSITION.INSTRUMENTAL.AZ.REFERENCED', '1.0');
ELSE
	fbComm.Publish('telescope', 'dome', 'POSITION.INSTRUMENTAL.AZ.REFERENCED', '0.0');
END_IF
//ERROR_STATE
IF fbAzimuth.Error THEN
	fbComm.Publish('telescope', 'dome', 'POSITION.INSTRUMENTAL.AZ.ERROR_STATE', UDINT_TO_STRING(fbAzimuth.ErrorID));
ELSE
	fbComm.Publish('telescope', 'dome', 'POSITION.INSTRUMENTAL.AZ.ERROR_STATE', '0');
END_IF
//MOTION_STATE
IF fbAzimuth.Busy THEN
	IF fbAzimuth.isTracking THEN
		fbComm.Publish('telescope', 'dome', 'POSITION.INSTRUMENTAL.AZ.MOTION_STATE', '8');
	ELSE
		fbComm.Publish('telescope', 'dome', 'POSITION.INSTRUMENTAL.AZ.MOTION_STATE', '1');
	END_IF
ELSE
	fbComm.Publish('telescope', 'dome', 'POSITION.INSTRUMENTAL.AZ.MOTION_STATE', '0');
END_IF

fbComm.Publish('telescope', 'dome', 'POSITION.INSTRUMENTAL.AZ.CURRPOS', LREAL_TO_STRING(fAzimuthCurrent));
fbComm.Publish('telescope', 'dome', 'POSITION.INSTRUMENTAL.AZ.REALPOS', LREAL_TO_STRING(fAzimuthCurrent-F_AzimuthOffsetOnAxis(fAzimuthOffset, fElevationCurrent)));	// M7: was fElevation (stale)
fbComm.Publish('telescope', 'dome', 'POSITION.INSTRUMENTAL.AZ.TARGETPOS', LREAL_TO_STRING(fbAzimuth.Position));
fbComm.Publish('telescope', 'dome', 'POSITION.INSTRUMENTAL.AZ.CURRSPEED', LREAL_TO_STRING(fbAzimuth.Velocity));
fbComm.Publish('telescope', 'dome', 'POSITION.INSTRUMENTAL.AZ.TARGETDISTANCE', LREAL_TO_STRING(ABS(fAzimuthCurrent-fbAzimuth.Position)));
fbComm.Publish('telescope', 'dome', 'POSITION.INSTRUMENTAL.AZ.OFFSET', LREAL_TO_STRING(fAzimuthOffset));


(*HORIZONTAL*)
fbComm.Publish('telescope', 'dome', 'POSITION.HORIZONTAL.ALT', LREAL_TO_STRING(fElevationCurrentSky));
fbComm.Publish('telescope', 'dome', 'POSITION.HORIZONTAL.AZ', LREAL_TO_STRING(fAzimuthCurrentSky));
//fbComm.Publish('telescope', 'dome', 'POSITION.HORIZONTAL.DOME', LREAL_TO_STRING(fbDome.Position));

(*EQUITORIAL*)
fbComm.Publish('telescope', 'dome', 'POSITION.EQUATORIAL.RA_ICRS', LREAL_TO_STRING(fRightAscensionCurrent));	// degrees (BROTLib#37)
fbComm.Publish('telescope', 'dome', 'POSITION.EQUATORIAL.HA_ICRS', LREAL_TO_STRING(fHourAngleCurrent));
fbComm.Publish('telescope', 'dome', 'POSITION.EQUATORIAL.DEC_ICRS', LREAL_TO_STRING(fDeclinationCurrent));
END_METHOD

METHOD PRIVATE _SlewTelescope : USINT
VAR_INPUT
END_VAR
VAR
	SlewEvent:	FB_Eventlog;
	command_timeout: TON;
END_VAR
VAR_STAT
	nStage:		USINT := 0;
	nLastStage:	USINT := 101;
END_VAR
_SlewTelescope := nStage;
command_timeout(IN := nStage < 100, PT := T#600S);
IF command_timeout.Q THEN
	bError := TRUE;
	nErrorID := 16#40;
	bSoftwareError := TRUE;
	nSoftwareErrorID := 16#40;
	bSlew := FALSE;
	nStage := 0;
	RETURN;
END_IF
IF bReset OR bError OR bInterrupted THEN
	nStage := 0;
	RETURN;
END_IF
CASE nStage OF
	0:	
		IF bReady AND bStopped AND NOT bBusy AND NOT bTracking THEN
			nStage := 10;
		END_IF
	10:
		IF fbElevation.Tracking = TRUE OR fbAzimuth.Tracking = TRUE OR fbDerotator.Tracking = TRUE THEN
			fbElevation.Tracking := FALSE;
			fbAzimuth.Tracking := FALSE;
			fbDerotator.Tracking := FALSE;
		ELSE
			nStage := 25;
		END_IF				
	25:
		fbPointing(
			fAzimuth			:= fAzimuth,
			fElevation			:= fElevation,
			fAzimuthOffset		=> fAzimuthPointingOffset,
			fElevationOffset	=> fElevationPointingOffset
		);	
		fbElevation.Position := fElevation + fElevationPointingOffset + fElevationOffset;
		fbElevation.Velocity := fElevationMoveVelocity;
		fbElevation.MoveAxis := TRUE;
		fbAzimuth.Position := fAzimuth + fAzimuthPointingOffset + F_AzimuthOffsetOnAxis(fAzimuthOffset, fElevation);	// M7: was fElevationCalc, mismatched with fAzimuth above
		fbAzimuth.Velocity := 10.0;
		fbAzimuth.MoveAxis := TRUE;
		fbDerotator.Position := fElevation + fDerotatorOffset;
		fbDerotator.Velocity := 10.0;
		fbDerotator.MoveAxis := TRUE;
		IF fbElevation.Busy AND
			fbAzimuth.Busy AND
			fbDerotator.Busy THEN
				nStage := 50;
		END_IF
	50:
		IF fbElevation.MoveDone THEN
			fbElevation.bMoveAxis := FALSE;
		END_IF
		
		IF fbAzimuth.MoveDone THEN
			fbAzimuth.MoveAxis := FALSE;
		END_IF

		IF fbDerotator.MoveDone THEN
			fbDerotator.MoveAxis := FALSE;
		END_IF
		IF NOT bSlewing AND bStopped THEN // all axis standstill
			nStage := 100;
		END_IF
	100:
		fbElevation.MoveAxis := FALSE;
		fbAzimuth.MoveAxis := FALSE;
		fbDerotator.MoveAxis := FALSE;
		fRightAscension := fRightAscensionCalc;
		fDeclination := fDeclinationCalc;
		bSlew := FALSE;
		nStage := 0;
END_CASE
SlewEvent(Trigger := nStage > nLastStage, FormatString := 'Slew progress: %s', OnMessage := USINT_TO_STRING(nStage), Comm := fbComm);
nLastStage := nStage;
END_METHOD

METHOD PRIVATE _StopTelescope : BOOL
VAR_INPUT
END_VAR
IF fbAzimuth.Tracking = TRUE OR fbElevation.Tracking = TRUE OR fbDerotator.Tracking = TRUE THEN
	fbAzimuth.Tracking := FALSE;
	fbElevation.Tracking := FALSE;
	fbDerotator.Tracking := FALSE;
ELSIF fbAzimuth.MoveAxis = TRUE OR  fbElevation.MoveAxis = TRUE OR fbDerotator.MoveAxis = TRUE THEN
	fbAzimuth.MoveAxis := FALSE;
	fbElevation.MoveAxis := FALSE;
	fbDerotator.MoveAxis := FALSE;
ELSE
	// Only issue Axis stop commands if they are moving
	IF NOT fbAzimuth.fbAxis.StandStill THEN
		fbAzimuth.StopAxis := TRUE;
	ELSE
		fbAzimuth.StopAxis := FALSE;
	END_IF
	
	IF NOT fbElevation.fbAxis.StandStill THEN
		fbElevation.StopAxis := TRUE;
	ELSE
		fbElevation.StopAxis := FALSE;
	END_IF	
	
	IF NOT fbDerotator.fbAxis.StandStill THEN
		fbDerotator.StopAxis := TRUE;
	ELSE
		fbDerotator.StopAxis := FALSE;
	END_IF	

	IF bStopped THEN
		fbAzimuth.StopAxis := FALSE;
		fbElevation.StopAxis := FALSE;
		fbDerotator.StopAxis := FALSE;
		_StopTelescope := FALSE;
	END_IF
END_IF
END_METHOD

METHOD PRIVATE _TrackTelescope : BOOL
VAR_INPUT
END_VAR
// Elevation
fDerotatorVelocity := F_Derotatorvelocity(fAzimuthCalc, fElevationCalc, telescopeConfig.latitude, fDerotatorSign);
fElevationVelocity := F_Elevationvelocity(fAzimuthCalc, telescopeConfig.latitude);
fAzimuthVelocity := F_Azimuthvelocity(fElevationCalc, fAzimuthCalc, telescopeConfig.latitude);
IF fElevationCurrent < 5.0 OR fElevationCurrent > 89.5 THEN
	bTrack := FALSE;
END_IF
IF fAzimuthCurrent > 440.0 THEN
	bTrack := FALSE;
END_IF
IF (fDerotatorCurrent < -69.0 AND fDerotatorVelocity<0.0) OR (fDerotatorCurrent > 379.0 AND fDerotatorVelocity>0.0) THEN
	bTrack := FALSE;
END_IF

fbElevation.Position := fElevationCalc;
IF NOT fbElevation.Tracking THEN
	fbElevation.Velocity := fElevationMoveVelocity;
	fbElevation.MoveAxis := TRUE;
	IF NOT fbElevation.Busy AND fbElevation.MoveDone THEN
		fbElevation.MoveAxis := FALSE;
		IF fbElevation.isTracking THEN
			fbElevation.Velocity := fElevationVelocity;
		ELSE
			fbElevation.Velocity := 3.0*fElevationVelocity;
		END_IF
		fbElevation.Velocity := fElevationVelocity;
		fbElevation.Tracking := TRUE;
	END_IF
ELSE
	fbElevation.Velocity := fElevationVelocity;
END_IF

// Azimuth
fbAzimuth.Position := fAzimuthCalc;
IF NOT fbAzimuth.Tracking THEN
	fbAzimuth.Velocity := 10.0;
	fbAzimuth.MoveAxis := TRUE;
	IF NOT fbAzimuth.Busy AND fbAzimuth.MoveDone THEN
		fbAzimuth.MoveAxis := FALSE;
		IF fbAzimuth.isTracking THEN
			fbAzimuth.Velocity := fAzimuthVelocity;
		ELSE
			fbAzimuth.Velocity := 3.0*fAzimuthVelocity;
		END_IF
		fbAzimuth.Velocity := fAzimuthVelocity;
		fbAzimuth.Tracking := TRUE;
	END_IF
ELSE
	fbAzimuth.Velocity := fAzimuthVelocity;
END_IF

// Derotator
fbDerotator.Position := fDerotatorCalc;
IF NOT fbDerotator.Tracking THEN
	fbDerotator.Velocity := 10.0;
	fbDerotator.MoveAxis := TRUE;
	IF NOT fbDerotator.Busy AND fbDerotator.MoveDone THEN
		fbDerotator.MoveAxis := FALSE;
		IF fbDerotator.isTracking THEN
			fbDerotator.Velocity := fDerotatorVelocity;
		ELSE
			fbDerotator.Velocity := 3.0*fDerotatorVelocity;
		END_IF
		fbDerotator.Velocity := fDerotatorVelocity;
		fbDerotator.Tracking := TRUE;
	END_IF
ELSE
	fbDerotator.Velocity := fDerotatorVelocity;
END_IF
END_METHOD

PROPERTY Altitude : LREAL
GET
Altitude := THIS^.fElevationCurrent;
END_GET
END_PROPERTY

PROPERTY Azimuth : LREAL
GET
Azimuth := THIS^.fAzimuthCurrent;
END_GET
END_PROPERTY

PROPERTY CoverAutoOpen : BOOL
GET
CoverAutoOpen := THIS^.bCoverAutoOpen;
END_GET
SET
// This property has no effect on MONET: _PowerOn always opens the covers
// unconditionally and never reads bCoverAutoOpen. Forcing it TRUE here keeps
// the property honest, but does not by itself guarantee the invariant, since
// bCoverAutoOpen is a public VAR_INPUT a caller can still write to directly.
THIS^.bCoverAutoOpen := TRUE;
END_SET
END_PROPERTY

PROPERTY Declination : LREAL
GET
Declination := THIS^.fDeclination;
END_GET
END_PROPERTY

METHOD Init : BOOL
bPower := TRUE;
END_METHOD

METHOD MoveAltAz : BOOL
VAR_INPUT
	AltAz	: BROTLib.ST_AltAzCoordinate;
END_VAR
fElevation 	:= AltAz.Altitude;
fAzimuth 	:= AltAz.Azimuth;
bSlew		:= TRUE;
END_METHOD

METHOD MoveRaDec : BOOL
VAR_INPUT
	RaDec	: BROTLib.ST_RaDecCoordinate;
END_VAR
fRightAscension	:= RaDec.RightAscension;
fDeclination	:= RaDec.Declination;
bGoto			:= TRUE;
END_METHOD

METHOD Park : BOOL
bPark := TRUE;
END_METHOD

METHOD Reset : BOOL
bReset := TRUE;
END_METHOD

PROPERTY RightAscension : LREAL
GET
RightAscension := THIS^.fRightAscension;
END_GET
END_PROPERTY

METHOD SetAltitudeOffset : BOOL
VAR_INPUT
	Offset	: LREAL;
END_VAR
fElevationOffset := Offset;
END_METHOD

METHOD SetAzimuthOffset : BOOL
VAR_INPUT
	Offset	: LREAL;
END_VAR
fAzimuthOffset := Offset;
END_METHOD

METHOD SetDerotatorOffset : BOOL
VAR_INPUT
	Offset	: LREAL;
END_VAR
fDerotatorOffset := Offset;
END_METHOD

METHOD Slew : BOOL
VAR_INPUT
	fAzimuth	: LREAL;
	fAltitude	: LREAL;
END_VAR
THIS^.fElevation 	:= fAltitude;
THIS^.fAzimuth 	:= fAzimuth;
THIS^.bSlew		:= TRUE;
END_METHOD

METHOD Stop : BOOL
bStop := TRUE;
END_METHOD

METHOD Track : BOOL
VAR_INPUT
	fRightAscension	: LREAL;
	fDeclination	: LREAL;
END_VAR
THIS^.fRightAscension	:= fRightAscension;
THIS^.fDeclination		:= fDeclination;
//THIS^.bTrack			:= TRUE;
THIS^.bGoto				:= TRUE;
END_METHOD

METHOD TrackRaDec : BOOL
VAR_INPUT
	RaDec	: BROTLib.ST_RaDecCoordinate;
END_VAR
fRightAscension	:= RaDec.RightAscension;
fDeclination		:= RaDec.Declination;
//bTrack			:= TRUE;
THIS^.bGoto				:= TRUE;
END_METHOD

END_FUNCTION_BLOCK

(* stored: Version 1.1.0.1, ProductVersion 3.1.4024.15
   POU FB_MonetTelescopeControl: Id {392c90d3-a441-4c8d-a752-42b25b49f5cd}, SpecialFunc None
   Folder internal methods: Id {d1e7fbc6-9662-4c16-bf25-8044ef92da3b}
   Method _GotoTelescope: Id {8976ce61-8856-40e1-8cfb-7b9454a4edbf}
   Method _HomeTelescope: Id {7bd4dae5-c49f-4cd9-a0c3-809697b8de19}
   Method _ParkTelescope: Id {999576b1-8aca-41eb-91ab-673a6fc7f4ba}
   Method _PowerOn: Id {4c40649f-56d9-4130-9f80-925439540d98}
   Method _SendTelemetry: Id {5e3ab35e-5dd6-4108-99df-8d99cebae004}
   Method _SlewTelescope: Id {d3e1cb80-5564-4d5b-b2d9-2c8dd1b9215a}
   Method _StopTelescope: Id {cb5cd062-03c6-4c9b-bbde-9c71b10960c3}
   Method _TrackTelescope: Id {6e849cc7-222d-486c-8d3d-ea253bc6d574}
   Property Altitude: Id {51b1ff05-1140-4331-8485-239187f5f8b1}
   Get Get: Id {05a6ac86-f3fe-4579-ad82-04708fa0864e}
   Property Azimuth: Id {0dd05217-329b-419a-a3b6-a7f2c3a7b182}
   Get Get: Id {fd6f0d71-0c53-4de5-af62-a6f082f3b2fe}
   Property CoverAutoOpen: Id {d750fe74-a7ce-44c0-a77d-2f5e342e939f}
   Get Get: Id {4134082f-796e-4360-8ca1-5611440c0e09}
   Set Set: Id {5af5b3f5-890f-4491-8b7f-06921498a3f2}
   Property Declination: Id {b1285964-102f-45b7-af05-6785154ef40d}
   Get Get: Id {add754b0-d14d-4a0e-b482-234fdfd51176}
   Method Init: Id {78ec73c4-02ac-4d83-aefd-694e0077d330}
   Method MoveAltAz: Id {94f5e9d8-f8f7-4c16-ac3f-2e854a5b373b}
   Method MoveRaDec: Id {86c89766-d350-4f6b-9fea-e302f9b4e7d4}
   Method Park: Id {21fb237d-ad50-4f82-97cf-a56a9c25b954}
   Method Reset: Id {efa0c84e-7359-43c3-a635-1faede103859}
   Property RightAscension: Id {11e4e9e9-9e18-4d9f-ab19-1c208929d2bc}
   Get Get: Id {b17aa26c-317b-4e3f-8426-b76a55e02df1}
   Method SetAltitudeOffset: Id {522d462f-4678-4f02-8df4-00f463761b00}
   Method SetAzimuthOffset: Id {16e0d010-c333-4c19-862e-702e715c040b}
   Method SetDerotatorOffset: Id {f59933b1-4aa9-4f18-88cf-26244adda0df}
   Method Slew: Id {ee4e9e45-2bba-488b-8094-f2bf4a28ec2b}
   Method Stop: Id {d33b3161-dc8a-45e5-ae2f-544550162c16}
   Method Track: Id {36f6a798-1a7b-442f-88f7-fc8d7dfa3dc0}
   Method TrackRaDec: Id {f497d99f-36a3-42c8-ae9b-738903f3158c} *)
